TYPE ST_STATE_TOUCH_PROBE :
STRUCT
  State           : UINT;   // 0 := deactivated, 100 := BUSY, 1000 := DONE, 9000 := ERROR
  LatchPositive   : LREAL;  // rising edge
  LatchNegative   : LREAL;  // falling edge
END_STRUCT
END_TYPE

(* stored: Version 1.1.0.1, ProductVersion 3.1.4024.13
   DUT ST_STATE_TOUCH_PROBE: Id {0b2fc911-fda9-407b-8cd6-cc279ae8d096} *)
